TYPE CM_Motor_HMI :
STRUCT
	Start		: BOOL;
	Stop		: BOOL;
	Reset		: BOOL;
	Abort		: BOOL;
	Clear		: BOOL;
	UnSuspend	: BOOL;
	Suspend		: BOOL;
	UnHold		: BOOL;
	Hold		: BOOL;
	Richting_L	: BOOL;
	Richting_R	: BOOL;
	Toerental	: INT;
	Auto		: BOOL;
	Manueel		: BOOL;
END_STRUCT
END_TYPE

(* stored: Version 1.1.0.1, ProductVersion 3.1.4024.12
   DUT CM_Motor_HMI: Id {cb87481b-20a4-44fd-8d06-ce7d47e19c4c} *)
